(* IEC 61131-3 sources: SafePLC-Gen-Evaluation/Evaluation Results/Dexpi_PDF/run_03, 2 files *)

(* ---- io_declarations.st ---- *)
(* ==================================================  *)
(* PLC I/O Variable Declarations — CODESYS 3.5  *)
(* Generated by SafePLC-Gen Multimodal  *)
(* ==================================================  *)

VAR_GLOBAL
    (* --- Analog Inputs ---  *)
    PI_4712.01_Raw               AT %IW0       : INT := 0;    (* PI-4712.01 — Pressure indicator, local, on line downs  *)
    PICSA_4712.02_Raw            AT %IW2       : INT := 0;    (* PICSA-4712.02 — Pressure indicator/controller/switch/ala  *)
    TICSA_4750.03_Raw            AT %IW4       : INT := 0;    (* TICSA-4750.03 — Temperature indicator/controller/switch/  *)
    (* --- Analog Outputs ---  *)
    FC_VALVE_H_1007_IN_Out       AT %QW0       : INT := 0;    (* FC-VALVE-H-1007-IN — Fail-closed (F.C.) control valve on line  *)
    PVA_4712.02_Out              AT %QW2       : INT := 0;    (* PVA-4712.02 — Pressure control valve A, tag PVA4712.02  *)
    TV_4750.03_Out               AT %QW4       : INT := 0;    (* TV-4750.03 — Temperature control valve, tag TV4750.03  *)
    (* --- Digital Inputs ---  *)
    HS_4750.01                   AT %IX0.0     : BOOL := FALSE;    (* HS-4750.01 — Hand switch / operator pushbutton statio  *)
    (* --- Digital Outputs ---  *)
    SV_104.01                    AT %QX0.0     : BOOL := FALSE;    (* SV-104.01 — Solenoid valve, tag SV 104.01, P=6 barg,  *)
END_VAR

(* ---- generated_code.st ---- *)
(* Generated by SafePLC-Gen Multimodal — CODESYS 3.5 *)
(* IEC 61131-3 Structured Text *)
(* Date: 2026-04-25T14:00:15.354757 *)

PROGRAM PressureTemperatureControl

VAR
    TICSA_4750_03_Raw            AT %IW4       : INT := 0;
    PICSA_4712_02_Raw            AT %IW2       : INT := 0;
    PI_4712_01_Raw               AT %IW0       : INT := 0;
    TV_4750_03_Out               AT %QW4       : INT := 0;
    PVA_4712_02_Out              AT %QW2       : INT := 0;
    FC_VALVE_H_1007_IN_Out       AT %QW0       : INT := 0;
    HS_4750_01                   AT %IX0.0     : BOOL := FALSE;
    SV_104_01                    AT %QX0.0     : BOOL := FALSE;
    ESTOP                        AT %IX0.1     : BOOL := FALSE;
    MANUAL_RESET                 AT %IX0.2     : BOOL := FALSE;
END_VAR

VAR
    TICSA_4750_03_Scaled         : REAL := 0.0;
    PICSA_4712_02_Scaled         : REAL := 0.0;
    PI_4712_01_Scaled            : REAL := 0.0;

    TICSA_4750_03_HH_SP          : REAL := 120.0;
    TICSA_4750_03_H_SP           : REAL := 110.0;
    TICSA_4750_03_L_SP           : REAL := 20.0;
    TICSA_4750_03_LL_SP          : REAL := 10.0;
    TICSA_4750_03_Deadband       : REAL := 2.0;

    PICSA_4712_02_HH_SP          : REAL := 9.0;
    PICSA_4712_02_H_SP           : REAL := 8.0;
    PICSA_4712_02_L_SP           : REAL := 1.0;
    PICSA_4712_02_LL_SP          : REAL := 0.5;
    PICSA_4712_02_Deadband       : REAL := 0.1;

    PI_4712_01_HH_SP             : REAL := 9.0;
    PI_4712_01_H_SP              : REAL := 8.0;
    PI_4712_01_L_SP              : REAL := 1.0;
    PI_4712_01_LL_SP             : REAL := 0.5;
    PI_4712_01_Deadband          : REAL := 0.1;

    TICSA_4750_03_HH             : BOOL := FALSE;
    TICSA_4750_03_H              : BOOL := FALSE;
    TICSA_4750_03_L              : BOOL := FALSE;
    TICSA_4750_03_LL             : BOOL := FALSE;
    TICSA_4750_03_HH_Ack         : BOOL := FALSE;
    TICSA_4750_03_LL_Ack         : BOOL := FALSE;
    TICSA_4750_03_HH_Set         : BOOL := FALSE;
    TICSA_4750_03_HH_Rst         : BOOL := FALSE;
    TICSA_4750_03_LL_Set         : BOOL := FALSE;
    TICSA_4750_03_LL_Rst         : BOOL := FALSE;
    TICSA_4750_03_HH_Latch       : SR := (S1 := FALSE, R := FALSE);
    TICSA_4750_03_LL_Latch       : SR := (S1 := FALSE, R := FALSE);

    PICSA_4712_02_HH             : BOOL := FALSE;
    PICSA_4712_02_H              : BOOL := FALSE;
    PICSA_4712_02_L              : BOOL := FALSE;
    PICSA_4712_02_LL             : BOOL := FALSE;
    PICSA_4712_02_HH_Ack         : BOOL := FALSE;
    PICSA_4712_02_LL_Ack         : BOOL := FALSE;
    PICSA_4712_02_HH_Set         : BOOL := FALSE;
    PICSA_4712_02_HH_Rst         : BOOL := FALSE;
    PICSA_4712_02_LL_Set         : BOOL := FALSE;
    PICSA_4712_02_LL_Rst         : BOOL := FALSE;
    PICSA_4712_02_HH_Latch       : SR := (S1 := FALSE, R := FALSE);
    PICSA_4712_02_LL_Latch       : SR := (S1 := FALSE, R := FALSE);

    PI_4712_01_HH                : BOOL := FALSE;
    PI_4712_01_H                 : BOOL := FALSE;
    PI_4712_01_L                 : BOOL := FALSE;
    PI_4712_01_LL                : BOOL := FALSE;
    PI_4712_01_HH_Ack            : BOOL := FALSE;
    PI_4712_01_LL_Ack            : BOOL := FALSE;
    PI_4712_01_HH_Set            : BOOL := FALSE;
    PI_4712_01_HH_Rst            : BOOL := FALSE;
    PI_4712_01_LL_Set            : BOOL := FALSE;
    PI_4712_01_LL_Rst            : BOOL := FALSE;
    PI_4712_01_HH_Latch          : SR := (S1 := FALSE, R := FALSE);
    PI_4712_01_LL_Latch          : SR := (S1 := FALSE, R := FALSE);

    LOOP_4750_03_TRIP            : BOOL := FALSE;
    LOOP_4712_02_TRIP            : BOOL := FALSE;
    SAFE_STATE                   : BOOL := FALSE;

    TICSA_4750_03_SP             : REAL := 80.0;
    TICSA_4750_03_Error          : REAL := 0.0;
    TICSA_4750_03_Integral       : REAL := 0.0;
    TICSA_4750_03_Kp             : REAL := 1.5;
    TICSA_4750_03_Ki             : REAL := 0.05;
    TICSA_4750_03_Output         : REAL := 0.0;

    PICSA_4712_02_SP             : REAL := 5.0;
    PICSA_4712_02_Error          : REAL := 0.0;
    PICSA_4712_02_Integral       : REAL := 0.0;
    PICSA_4712_02_Kp             : REAL := 2.0;
    PICSA_4712_02_Ki             : REAL := 0.08;
    PICSA_4712_02_Output         : REAL := 0.0;

    FC_VALVE_Output              : REAL := 0.0;
    System_Alarm                 : BOOL := FALSE;
    FirstScan                    : BOOL := TRUE;
END_VAR

IF FirstScan THEN
    LOOP_4750_03_TRIP      := TRUE;
    LOOP_4712_02_TRIP      := TRUE;
    SAFE_STATE             := TRUE;
    TV_4750_03_Out         := 6554;
    PVA_4712_02_Out        := 6554;
    FC_VALVE_H_1007_IN_Out := 6554;
    SV_104_01              := FALSE;
    FirstScan              := FALSE;
    RETURN;
END_IF;

TICSA_4750_03_Scaled := ((INT_TO_REAL(TICSA_4750_03_Raw) - 6554.0) / (32767.0 - 6554.0)) * 150.0;
PICSA_4712_02_Scaled := ((INT_TO_REAL(PICSA_4712_02_Raw) - 6554.0) / (32767.0 - 6554.0)) * 10.0;
PI_4712_01_Scaled    := ((INT_TO_REAL(PI_4712_01_Raw)    - 6554.0) / (32767.0 - 6554.0)) * 10.0;

IF TICSA_4750_03_Scaled >= TICSA_4750_03_HH_SP THEN
    TICSA_4750_03_HH_Set := TRUE;
ELSIF TICSA_4750_03_Scaled <= (TICSA_4750_03_HH_SP - TICSA_4750_03_Deadband) THEN
    TICSA_4750_03_HH_Set := FALSE;
END_IF;
TICSA_4750_03_HH_Rst := TICSA_4750_03_HH_Ack AND (TICSA_4750_03_Scaled < TICSA_4750_03_HH_SP);
TICSA_4750_03_HH_Latch(S1 := TICSA_4750_03_HH_Set, R := TICSA_4750_03_HH_Rst);
TICSA_4750_03_HH := TICSA_4750_03_HH_Latch.Q1;

TICSA_4750_03_H := TICSA_4750_03_Scaled >= TICSA_4750_03_H_SP;
TICSA_4750_03_L := TICSA_4750_03_Scaled <= TICSA_4750_03_L_SP;

IF TICSA_4750_03_Scaled <= TICSA_4750_03_LL_SP THEN
    TICSA_4750_03_LL_Set := TRUE;
ELSIF TICSA_4750_03_Scaled >= (TICSA_4750_03_LL_SP + TICSA_4750_03_Deadband) THEN
    TICSA_4750_03_LL_Set := FALSE;
END_IF;
TICSA_4750_03_LL_Rst := TICSA_4750_03_LL_Ack AND (TICSA_4750_03_Scaled > TICSA_4750_03_LL_SP);
TICSA_4750_03_LL_Latch(S1 := TICSA_4750_03_LL_Set, R := TICSA_4750_03_LL_Rst);
TICSA_4750_03_LL := TICSA_4750_03_LL_Latch.Q1;

IF PICSA_4712_02_Scaled >= PICSA_4712_02_HH_SP THEN
    PICSA_4712_02_HH_Set := TRUE;
ELSIF PICSA_4712_02_Scaled <= (PICSA_4712_02_HH_SP - PICSA_4712_02_Deadband) THEN
    PICSA_4712_02_HH_Set := FALSE;
END_IF;
PICSA_4712_02_HH_Rst := PICSA_4712_02_HH_Ack AND (PICSA_4712_02_Scaled < PICSA_4712_02_HH_SP);
PICSA_4712_02_HH_Latch(S1 := PICSA_4712_02_HH_Set, R := PICSA_4712_02_HH_Rst);
PICSA_4712_02_HH := PICSA_4712_02_HH_Latch.Q1;

PICSA_4712_02_H := PICSA_4712_02_Scaled >= PICSA_4712_02_H_SP;
PICSA_4712_02_L := PICSA_4712_02_Scaled <= PICSA_4712_02_L_SP;

IF PICSA_4712_02_Scaled <= PICSA_4712_02_LL_SP THEN
    PICSA_4712_02_LL_Set := TRUE;
ELSIF PICSA_4712_02_Scaled >= (PICSA_4712_02_LL_SP + PICSA_4712_02_Deadband) THEN
    PICSA_4712_02_LL_Set := FALSE;
END_IF;
PICSA_4712_02_LL_Rst := PICSA_4712_02_LL_Ack AND (PICSA_4712_02_Scaled > PICSA_4712_02_LL_SP);
PICSA_4712_02_LL_Latch(S1 := PICSA_4712_02_LL_Set, R := PICSA_4712_02_LL_Rst);
PICSA_4712_02_LL := PICSA_4712_02_LL_Latch.Q1;

IF PI_4712_01_Scaled >= PI_4712_01_HH_SP THEN
    PI_4712_01_HH_Set := TRUE;
ELSIF PI_4712_01_Scaled <= (PI_4712_01_HH_SP - PI_4712_01_Deadband) THEN
    PI_4712_01_HH_Set := FALSE;
END_IF;
PI_4712_01_HH_Rst := PI_4712_01_HH_Ack AND (PI_4712_01_Scaled < PI_4712_01_HH_SP);
PI_4712_01_HH_Latch(S1 := PI_4712_01_HH_Set, R := PI_4712_01_HH_Rst);
PI_4712_01_HH := PI_4712_01_HH_Latch.Q1;

PI_4712_01_H := PI_4712_01_Scaled >= PI_4712_01_H_SP;
PI_4712_01_L := PI_4712_01_Scaled <= PI_4712_01_L_SP;

IF PI_4712_01_Scaled <= PI_4712_01_LL_SP THEN
    PI_4712_01_LL_Set := TRUE;
ELSIF PI_4712_01_Scaled >= (PI_4712_01_LL_SP + PI_4712_01_Deadband) THEN
    PI_4712_01_LL_Set := FALSE;
END_IF;
PI_4712_01_LL_Rst := PI_4712_01_LL_Ack AND (PI_4712_01_Scaled > PI_4712_01_LL_SP);
PI_4712_01_LL_Latch(S1 := PI_4712_01_LL_Set, R := PI_4712_01_LL_Rst);
PI_4712_01_LL := PI_4712_01_LL_Latch.Q1;

IF TICSA_4750_03_HH OR TICSA_4750_03_LL THEN
    LOOP_4750_03_TRIP := TRUE;
ELSIF LOOP_4750_03_TRIP AND MANUAL_RESET
      AND NOT TICSA_4750_03_HH AND NOT TICSA_4750_03_LL THEN
    LOOP_4750_03_TRIP := FALSE;
END_IF;

IF PICSA_4712_02_HH OR PICSA_4712_02_LL THEN
    LOOP_4712_02_TRIP := TRUE;
ELSIF LOOP_4712_02_TRIP AND MANUAL_RESET
      AND NOT PICSA_4712_02_HH AND NOT PICSA_4712_02_LL THEN
    LOOP_4712_02_TRIP := FALSE;
END_IF;

SAFE_STATE := ESTOP OR LOOP_4750_03_TRIP OR LOOP_4712_02_TRIP;

IF NOT SAFE_STATE THEN
    TICSA_4750_03_Error    := TICSA_4750_03_SP - TICSA_4750_03_Scaled;
    TICSA_4750_03_Integral := TICSA_4750_03_Integral + (TICSA_4750_03_Ki * TICSA_4750_03_Error);
    IF TICSA_4750_03_Integral > 100.0 THEN
        TICSA_4750_03_Integral := 100.0;
    ELSIF TICSA_4750_03_Integral < 0.0 THEN
        TICSA_4750_03_Integral := 0.0;
    END_IF;
    TICSA_4750_03_Output := (TICSA_4750_03_Kp * TICSA_4750_03_Error) + TICSA_4750_03_Integral;
    IF TICSA_4750_03_Output > 100.0 THEN
        TICSA_4750_03_Output := 100.0;
    ELSIF TICSA_4750_03_Output < 0.0 THEN
        TICSA_4750_03_Output := 0.0;
    END_IF;
    TV_4750_03_Out := REAL_TO_INT(6554.0 + (TICSA_4750_03_Output / 100.0) * (32767.0 - 6554.0));
ELSE
    TV_4750_03_Out := 6554;
END_IF;

IF NOT SAFE_STATE THEN
    PICSA_4712_02_Error    := PICSA_4712_02_SP - PICSA_4712_02_Scaled;
    PICSA_4712_02_Integral := PICSA_4712_02_Integral + (PICSA_4712_02_Ki * PICSA_4712_02_Error);
    IF PICSA_4712_02_Integral > 100.0 THEN
        PICSA_4712_02_Integral := 100.0;
    ELSIF PICSA_4712_02_Integral < 0.0 THEN
        PICSA_4712_02_Integral := 0.0;
    END_IF;
    PICSA_4712_02_Output := (PICSA_4712_02_Kp * PICSA_4712_02_Error) + PICSA_4712_02_Integral;
    IF PICSA_4712_02_Output > 100.0 THEN
        PICSA_4712_02_Output := 100.0;
    ELSIF PICSA_4712_02_Output < 0.0 THEN
        PICSA_4712_02_Output := 0.0;
    END_IF;
    PVA_4712_02_Out := REAL_TO_INT(6554.0 + (PICSA_4712_02_Output / 100.0) * (32767.0 - 6554.0));
ELSE
    PVA_4712_02_Out := 6554;
END_IF;

IF NOT SAFE_STATE THEN
    IF HS_4750_01 THEN
        FC_VALVE_Output := 100.0;
    ELSE
        FC_VALVE_Output := 0.0;
    END_IF;
    FC_VALVE_H_1007_IN_Out := REAL_TO_INT(6554.0 + (FC_VALVE_Output / 100.0) * (32767.0 - 6554.0));
ELSE
    FC_VALVE_H_1007_IN_Out := 6554;
END_IF;

SV_104_01 := NOT SAFE_STATE;

System_Alarm :=
    TICSA_4750_03_HH_Latch.Q1 OR TICSA_4750_03_LL_Latch.Q1 OR
    TICSA_4750_03_H            OR TICSA_4750_03_L            OR
    PICSA_4712_02_HH_Latch.Q1 OR PICSA_4712_02_LL_Latch.Q1 OR
    PICSA_4712_02_H            OR PICSA_4712_02_L            OR
    PI_4712_01_HH_Latch.Q1    OR PI_4712_01_LL_Latch.Q1    OR
    PI_4712_01_H               OR PI_4712_01_L              OR
    LOOP_4750_03_TRIP          OR LOOP_4712_02_TRIP         OR
    SAFE_STATE;

END_PROGRAM
